{attribute addProperty BoxType "EL9210-0000-0016"}
{attribute addProperty Id "FuseErrorAT %I*BOOL81"}
{attribute addProperty CRC "1047352275"}
{attribute addProperty SizeInBites "8"}
{attribute addProperty SizeInBytes "1"}
TYPE FuseError_3E6D53D3 :
STRUCT
	{attribute addProperty Name "FuseError"}
	FuseError AT %I* : BOOL;
END_STRUCT
END_TYPE

(* stored: Version 1.2.0.0, ProductVersion 3.1.4024.9
   DUT FuseError_3E6D53D3: Id {e2aea739-b09e-421d-9ffd-6799a96bfdad} *)
